Fanuc KAREL source: kt00150.KL

-- PROVISIONAL review KL for V770-1; original PC SHA256 d3a3542cb1c8ca1d85817badc532be0b4b5ebce3cee30078cd0800e094266770
-- Incomplete behavior may be omitted. Consult companion uncertainty JSON. Do not deploy.
PROGRAM KT00150
%NOLOCKGROUP
VAR
  OUT : REAL
-- UNRESOLVED_DECL Y1 type=002018
-- UNRESOLVED_DECL Y2 type=002018
BEGIN
  -- UNRESOLVED_PC offsets 5-19; opcodes 2E,22,9D,33,B2
  -- UNRESOLVED_PC offsets 24-38; opcodes 2E,22,9D,33,B2
  -- UNRESOLVED_PC offsets 43-57; opcodes 2E,22,9D,33,B2
  -- UNRESOLVED_PC offsets 62-76; opcodes 2E,22,9D,33,B2
  -- UNRESOLVED_PC offsets 81-107; opcodes 22,9D,33,B1,22,9D,33,B1,55,64,23
  -- UNRESOLVED_PC offsets 112-116; opcodes 7F
END KT00150
